(* IEC 61131-3 sources: AXOpen/src/TestSandbox/ctrl/src/TestedControlUnit/Data, 4 files *)

(* ---- ScrewData.st ---- *)
NAMESPACE sandboxtest.StandardControlUnit
    USING AXOpen.Core;
    USING System.Strings;

TYPE ScrewData : STRUCT
            // {#ix-set:AttributeName = "Screw data"}
        // {#ix-attr:[Container(Layout.Stack)]}
        // {#ix-attr:[Group(GroupLayout.GroupBox)]}
        Result : AXOpen.Inspectors.AxoDigitalInspector;
        Torque : AXOpen.Inspectors.AxoAnalogueInspector;
        Angle : AXOpen.Inspectors.AxoAnalogueInspector;
        XCoordination : AXOpen.Inspectors.AxoAnalogueInspector;
        YCoordination : AXOpen.Inspectors.AxoAnalogueInspector;
    END_STRUCT;
END_TYPE

END_NAMESPACE

(* ---- FragmentProcessData.st ---- *)
NAMESPACE sandboxtest.StandardControlUnit
    USING AXOpen.Core;
    USING System.Strings;

    {#ix-attr:[Container(Layout.Tabs)]}
    CLASS FragmentProcessData
        EXTENDS AXOpen.Data.AxoDataEntity
        VAR PUBLIC
            CounterDelay : ULINT;
            // Screw_0 : sandboxtest.StandardControlUnit.ScrewData;
            // Screw_1 : sandboxtest.StandardControlUnit.ScrewData;
            // Screw_2 : sandboxtest.StandardControlUnit.ScrewData;
            // Screw_3 : sandboxtest.StandardControlUnit.ScrewData;
            // Screw_4 : sandboxtest.StandardControlUnit.ScrewData;

            Res_Screw_0 : AXOpen.Inspectors.AxoDigitalInspector;
            Tor_Screw_0 : AXOpen.Inspectors.AxoAnalogueInspector;
            Ang_Screw_0 : AXOpen.Inspectors.AxoAnalogueInspector;
            XCo_Screw_0 : AXOpen.Inspectors.AxoAnalogueInspector;
            YCo_Screw_0 : AXOpen.Inspectors.AxoAnalogueInspector;

            Res_Screw_1 : AXOpen.Inspectors.AxoDigitalInspector;
            Tor_Screw_1 : AXOpen.Inspectors.AxoAnalogueInspector;
            Ang_Screw_1 : AXOpen.Inspectors.AxoAnalogueInspector;
            XCo_Screw_1 : AXOpen.Inspectors.AxoAnalogueInspector;
            YCo_Screw_1 : AXOpen.Inspectors.AxoAnalogueInspector;

            Res_Screw_2 : AXOpen.Inspectors.AxoDigitalInspector;
            Tor_Screw_2 : AXOpen.Inspectors.AxoAnalogueInspector;
            Ang_Screw_2 : AXOpen.Inspectors.AxoAnalogueInspector;
            XCo_Screw_2 : AXOpen.Inspectors.AxoAnalogueInspector;
            YCo_Screw_2 : AXOpen.Inspectors.AxoAnalogueInspector;

            Res_Screw_3 : AXOpen.Inspectors.AxoDigitalInspector;
            Tor_Screw_3 : AXOpen.Inspectors.AxoAnalogueInspector;
            Ang_Screw_3 : AXOpen.Inspectors.AxoAnalogueInspector;
            XCo_Screw_3 : AXOpen.Inspectors.AxoAnalogueInspector;
            YCo_Screw_3 : AXOpen.Inspectors.AxoAnalogueInspector;

            Res_Screw_4 : AXOpen.Inspectors.AxoDigitalInspector;
            Tor_Screw_4 : AXOpen.Inspectors.AxoAnalogueInspector;
            Ang_Screw_4 : AXOpen.Inspectors.AxoAnalogueInspector;
            XCo_Screw_4 : AXOpen.Inspectors.AxoAnalogueInspector;
            YCo_Screw_4 : AXOpen.Inspectors.AxoAnalogueInspector;

            Traca__0 : AXOpen.Inspectors.AxoDataInspector;
            Traca__1 : AXOpen.Inspectors.AxoDataInspector;
            Reader_0 : AXOpen.Inspectors.AxoDataInspector;
            Reader_1 : AXOpen.Inspectors.AxoDataInspector;
            Camera_0 : AXOpen.Inspectors.AxoDataInspector;
            Camera_1 : AXOpen.Inspectors.AxoDataInspector;
        END_VAR
    END_CLASS

END_NAMESPACE

(* ---- FragmentProcessDataManger.st ---- *)
NAMESPACE sandboxtest.StandardControlUnit
    USING AXOpen.Core;
    USING System.Strings;
    USING AXOpen.Cognex.Vision.v_6_0_0_0;
    USING AXOpen.Elements;

    CLASS FragmentProcessDataManger
        EXTENDS AXOpen.Data.AxoDataExchange
        VAR PUBLIC
            {#ix-generic:TOnline}
            {#ix-generic:TPlain as POCO}
            {#ix-attr:[AXOpen.Data.AxoDataEntityAttribute]}
            {#ix-attr:[Container(Layout.Stack)]}
            {#ix-set:AttributeName = "Cux"}
            Set : FragmentProcessData;
        END_VAR
    END_CLASS

END_NAMESPACE

(* ---- ProcessDataManger.st ---- *)
NAMESPACE sandboxtest.StandardControlUnit
    USING AXOpen.Core;
    USING System.Strings;
    USING AXOpen.Cognex.Vision.v_6_0_0_0;

    CLASS ProcessDataManger
        EXTENDS AXOpen.Data.AxoDataFragmentExchange
        VAR PUBLIC
            {#ix-attr:[AXOpen.Data.AxoDataFragmentAttribute]}
            Shared : SharedProductionDataManager;
            {#ix-attr:[AXOpen.Data.AxoDataFragmentAttribute]}
            DataManger : FragmentProcessDataManger;
        END_VAR
    END_CLASS

END_NAMESPACE
